{attribute addProperty BoxType "EL7041-0000-0016"}
{attribute addProperty Id "ENC_Status_compactAT %I*ENC_Status_compact_58C6E2B94860STM_StatusAT %I*STM_Status_C2B0CAE11620ENC_Control_compactAT %Q*ENC_Control_compact_03701F333240STM_ControlAT %Q*STM_Control_6F24B2C41620STM_VelocityAT %Q*STM_Velocity_1D89B5C21620WcStateAT %I*WcState_98A4DF7520.250InfoDataAT %I*InfoData_6C7DEEF988110"}
{attribute addProperty CRC "2084361319"}
{attribute addProperty SizeInBites "218"}
{attribute addProperty SizeInBytes "27.25"}
TYPE EL7041_F90A6389 :
STRUCT
	{attribute addProperty Name "ENC_Status_compact"}
	ENC_Status_compact : ENC_Status_compact_58C6E2B9;
	{attribute addProperty Name "STM_Status"}
	STM_Status : STM_Status_C2B0CAE1;
	{attribute addProperty Name "ENC_Control_compact"}
	ENC_Control_compact : ENC_Control_compact_03701F33;
	{attribute addProperty Name "STM_Control"}
	STM_Control : STM_Control_6F24B2C4;
	{attribute addProperty Name "STM_Velocity"}
	STM_Velocity : STM_Velocity_1D89B5C2;
	{attribute addProperty Name "WcState"}
	WcState : WcState_98A4DF75;
	{attribute addProperty Name "InfoData"}
	InfoData : InfoData_6C7DEEF9;
END_STRUCT
END_TYPE

(* stored: Version 1.2.0.0, ProductVersion 3.1.4024.9
   DUT EL7041_F90A6389: Id {fef9dcb0-a472-44f4-94e5-f4ddc4aee103} *)
